# B&R Automation Studio project RTFProj (part 3)

#### Bar_light.c
```c
#include <bur/plctypes.h>
#include <MTBasics.h>
#include <brsystem.h>
#include <math.h>

#ifdef _DEFAULT_INCLUDES
#include <AsDefault.h>
#endif

void resetFB(struct Light *inst);												//Reset basic variables
void PWMControl(struct Light *inst);											//Controls Light in PWM Mode
void BlinkControl(struct Light *inst);											//Allows Blinking of Light

void Light(struct Light *inst)
{
	if ((!inst->Enable) && (inst->internal.MainControlBarLight != INIT_BARLIGHT))//If FB not allowed and switch is not in init state
		inst->internal.MainControlBarLight = DISABLED_BARLIGHT;					//Change state to DISABLED

	switch (inst->internal.MainControlBarLight)									//Main switch controls whole FB
	{
		case INIT_BARLIGHT:														//Check parameter for PWM
			inst->internal.TaskClass.RTInfo_0.enable = 1;
			RTInfo(&inst->internal.TaskClass.RTInfo_0);
			if (!(inst->internal.TaskClass.RTInfo_0.status) && (inst->internal.TaskClass.RTInfo_0.cycle_time > 0))
			{
				if (inst->internal.TaskClass.RTInfo_0.cycle_time <= 1000)
				{
					inst->isPWMEnabled = inst->internal.PWM.PWMEnabled = 1;
					inst->isPWMEnabled = inst->internal.PWM.PWM.Enable = 1;
					inst->internal.PWM.PWM.MinPulseWidth = 0.0008;
					inst->internal.PWM.PWM.Period = 0.008;
					inst->internal.PWM.PWM.Mode = mtBASICS_PULSE_BEGINNING;
				}
				else
					inst->isPWMEnabled = inst->internal.PWM.PWMEnabled = 0;

				inst->internal.PWM.PWM.DutyCycle = 100;
				inst->internal.TaskClass.RTInfo_0.enable = 0;
				inst->internal.TaskClass.CyclicTime = ((inst->internal.TaskClass.RTInfo_0.cycle_time)/800);
				inst->internal.MainControlBarLight = DISABLED_BARLIGHT;
			}
			break;

		case DISABLED_BARLIGHT:
			if (inst->Enable)
			{
				if (inst->DO9322.ModuleOK)
				{
					inst->internal.MainControlBarLight = ENABLED_BARLIGHT;
					resetFB(inst);
				}
				else
				{
					inst->Status = DO9322_NOT_CONNECTED;
					inst->internal.MainControlBarLight = ERROR_BARLIGHT;
				}
			}
			inst->isPowerOn = 0;
			break;

		case ENABLED_BARLIGHT:
			inst->Active = 1;
			if (inst->PowerOn)
			{
				if (inst->Blinking.StartBlinking)
				{
					BlinkControl(inst);
				}
				else if (inst->internal.PWM.PWMEnabled)
				{
					PWMControl(inst);
				}
				else inst->DO9322.DigitalOutput = 1;
				inst->isPowerOn = 1;
			}

			else{
				inst->DO9322.DigitalOutput = 0;
				inst->isPowerOn = 0;
			}
			break;

		case ERROR_BARLIGHT:
			inst->Error = 1;
			break;
	}
}

void resetFB(struct Light *inst)
{
	inst->Active = 0;
	inst->Blinking.StartBlinking = 0;
	inst->DO9322.DigitalOutput = 0;
	inst->DutyCycle = 100;
	inst->Error = 0;
	inst->isPowerOn = 0;
	inst->Status = ERR_OK;
}

void PWMControl(struct Light *inst)
{
	inst->internal.PWM.PWM.DutyCycle = inst->DutyCycle;
	MTBasicsPWM(&inst->internal.PWM.PWM);
	inst->DO9322.DigitalOutput = inst->internal.PWM.PWM.Out;
}

void BlinkControl(struct Light *inst)
{
	inst->internal.BlinkingCounter += 1;
	if ((inst->internal.BlinkingCounter*inst->internal.TaskClass.CyclicTime) < inst->Blinking.BlinkingTime_ms)
	{
		if ((inst->internal.BlinkCounter*inst->internal.TaskClass.CyclicTime) >= inst->Blinking.BlinkPeriod_ms)
		{
			inst->DO9322.DigitalOutput = !inst->DO9322.DigitalOutput;
			inst->internal.BlinkCounter = 0;
		}
		else
		{
			inst->internal.BlinkCounter += 1;
		}
	}
	else
	{
		inst->internal.BlinkingCounter = 0;
		inst->internal.BlinkCounter = 0;
		inst->DO9322.DigitalOutput = 0;
		inst->Blinking.StartBlinking = 0;
	}
}
```

#### Types.typ - Exported data types
```iecst
TYPE
	MainControlBarLight_enum :
		(
		INIT_BARLIGHT := 0,
		DISABLED_BARLIGHT := 1,
		ENABLED_BARLIGHT := 2,
		ERROR_BARLIGHT := 100
		);
	DO9322_type : 	STRUCT
		ModuleOK : BOOL;
		DigitalOutput : BOOL;
	END_STRUCT;
	PWM_type : 	STRUCT
		PWMEnabled : BOOL;
		PWM : MTBasicsPWM;
	END_STRUCT;
	internal_type : 	STRUCT
		init : BOOL;
		TaskClass : TaskClass_type;
		PWM : PWM_type;
		BlinkTime : UINT;
		MainControlBarLight : MainControlBarLight_enum;
		BlinkingCounter : UINT;
		BlinkCounter : UINT;
	END_STRUCT;
	Blink_type : 	STRUCT
		StartBlinking : BOOL;
		BlinkPeriod_ms : UINT;
		BlinkingTime_ms : UINT;
	END_STRUCT;
	TaskClass_type : 	STRUCT
		CyclicTime : UINT;
		RTInfo_0 : RTInfo;
	END_STRUCT;
END_TYPE
```

#### Constants.var - Exported constants
```iecst
VAR CONSTANT
	DO9322_NOT_CONNECTED : UINT := 62150; (*DO module in not connected*)
END_VAR
```

#### Bar_Light.fun - Exported functions and function blocks
```iecst
FUNCTION_BLOCK Light
	VAR_INPUT
		Enable : BOOL;
		DO9322 : DO9322_type;
		PowerOn : BOOL;
		DutyCycle : USINT; (*Power of Light in % [0-100]*)
		Blinking : Blink_type;
	END_VAR
	VAR_OUTPUT
		Active : BOOL;
		Error : BOOL;
		Status : UINT;
		isPWMEnabled : BOOL;
		isPowerOn : BOOL;
	END_VAR
	VAR
		internal : internal_type;
	END_VAR
END_FUNCTION_BLOCK
```

### Data object Logical/ACP10_ETXEN/acp10etxen (Ett)

- acp10etxen.ett (not shown)

### Program Logical/Simulation/Technology/simulation (ANSIC) - Roman Parák program for simulation.

#### simulation.c - Init, cyclic, exit code
```c
/*********************************************************************************************
* B&R Automation - Perfection in Automation (https://www.br-automation.com)
    ******************************************************************************************
    * Program 	    : Master's Thesis - Soccer Table (Simulation)
    * Author  	    : Roman Parak
    * Created 	    : date ...
	* University    : Brno University of Technology(BUT)
	* Faculty       : Faculty of Mechanical Engineering(FME)
	* Study Program : Applied Computer Science and Control
	* Institute     : Institute of Automation and Computer Science
**********************************************************************************************
* Implementation OF PROGRAM simulation(Simulation/Technology/simulation/Program/simulation.c)
**********************************************************************************************/

/*************************** LIBRARIES *********************************/
#include <bur/plc.h>
#include <bur/plctypes.h>
#include <astime.h>
#include <math.h>

#include "rp_funcx1.h"
#include "Structures/simulation_str.h"
#include "Functions/sim_mapp.h"

#ifdef _DEFAULT_INCLUDES
	#include <AsDefault.h>
#endif

/*************************** DEFINITIONS *******************************/
#define EACH_FORMATION 1;

/************************ LOCAL VARIABLES ******************************/

// struct - rp_funcx1
_LOCAL struct forecast_direction f_d;
_LOCAL struct calculation_posDummies c_ppd;
_LOCAL struct calculation_crossingBall c_cb[2];
_LOCAL struct calculation_displacementOfAxes c_doa;
_LOCAL struct start_rotaryAxis start_rotaryAxis_0;
_LOCAL struct control_temperature c_temp;
_LOCAL struct axes_control axes_control_0[4];
_LOCAL struct ball_shooting ball_s;
_LOCAL struct check_attack_mode check_attack_mode_0;
_LOCAL struct start_virtualAxis s_virtualA;
// struct - MpAlarmX
_LOCAL MpAlarmXListUIConnectType AlarmListUI_ConnectType;
_LOCAL MpAlarmXHistoryUIConnectType AlarmHistoryUI_ConnectType;
// udint
_LOCAL UDINT alarm_device_address, specific_directionOfBall;
// usint
_LOCAL USINT max_numberOfFormation;
_LOCAL USINT i_axisNum;
_LOCAL USINT i_bs;
_LOCAL USINT i_ppd, i_ccd, i_ccdCPU, i_ccdHUM, i_cdoa1, i_cdoa2, i_cdoa3;
_LOCAL USINT c_dp;
_LOCAL USINT i_def, i_dp1, i_dp2;
_LOCAL USINT c_bState;
// bool
_LOCAL BOOL ESTOP,error_s,reset_safetyESTOP;
_LOCAL BOOL start_game;
// real
_LOCAL REAL x_posOfCPU[4];
_LOCAL REAL x_posOfHUM[4];
// OUPTUT from the SENSOR & CAMERA
_LOCAL REAL ball1[2], ball2[2], time_B2B;
_LOCAL REAL optical_sensor[4];
_LOCAL REAL reflex_sensor[4];
// state machine
_LOCAL soccer_table_ENUM SOCCER_TABLE_STEP;
_LOCAL soccer_table_ENUM BEFORE_STATE;

/**********************************************************************************************************/
/********************************************** INIT PROGRAM **********************************************/
/**********************************************************************************************************/
void _INIT ProgramInit(void)
{
    /*********************************** declaration variables **********************************/
    // generally
    max_numberOfFormation = 4;
    // axis type -> MAPP
    // linear
	gLinkAxes_linear[0] = gk_mappAxisLS;
    gLinkAxes_linear[1] = df_mappAxisLS;
    gLinkAxes_linear[2] = md_mappAxisLS;
    gLinkAxes_linear[3] = fw_mappAxisLS;
    // rotary
    gLinkAxes_rotary[0] = gk_mappAxisRS;
    gLinkAxes_rotary[1] = df_mappAxisRS;
    gLinkAxes_rotary[2] = md_mappAxisRS;
    gLinkAxes_rotary[3] = fw_mappAxisRS;

    /************************************ control of AlarmX ************************************/
    // adjustment device name
    alarm_device_address = (UDINT) strcpy(mp_alarmX.deviceName_no1_exp,"EXPORT_HISTORY");
    // MpAlarmX Core
    mp_alarmX.mp_core.MpLink         = &gAlarmXCoreS;
    mp_alarmX.mp_core.Enable         = 1;
    // MpAlarmX ListUI
    mp_alarmX.mp_listUI.MpLink       = &gAlarmXCoreS;
    mp_alarmX.mp_listUI.Enable       = 1;
    mp_alarmX.mp_listUI.UIConnect    = &AlarmListUI_ConnectType;
    // MpAlarmX History
    mp_alarmX.mp_history.MpLink      = &gAlarmXHistoryS;
    mp_alarmX.mp_history.Enable      = 1;
    mp_alarmX.mp_history.DeviceName  = &mp_alarmX.deviceName_no1_exp;
    // MpAlarmX HistoryUI
    mp_alarmX.mp_historyUI.MpLink    = &gAlarmXHistoryS;
    mp_alarmX.mp_historyUI.Enable    = 1;
    mp_alarmX.mp_historyUI.UIConnect = &AlarmHistoryUI_ConnectType;

    /************************************* control of axes **************************************/
    for(i_axisNum = 0; i_axisNum <= max_numberOfFormation - 1; i_axisNum++){
        // initialization ACOPOS variables through function(get_axisParam), that returns two variables type of UDINT
        // into the structure -> axesAcopos(have two parameters : linear, rotary)
        axis_acopos = get_axisParam(i_axisNum);
        // linear -> LinMot
        // linear axis basic
        mp_Axis.mp_axisLinear[i_axisNum].Enable     = 1;
        mp_Axis.mp_axisLinear[i_axisNum].MpLink     = &gLinkAxes_linear[i_axisNum];
        mp_Axis.mp_axisLinear[i_axisNum].Parameters = &mp_Axis.param_axisLinear[i_axisNum];
        mp_Axis.mp_axisLinear[i_axisNum].Axis       = axis_acopos.linear;
        // linear cyclic set
        mp_Axis.mp_cyclicSetLinear[i_axisNum].Enable     = 1;
        mp_Axis.mp_cyclicSetLinear[i_axisNum].MpLink     = &gLinkAxes_linear[i_axisNum];
        mp_Axis.mp_cyclicSetLinear[i_axisNum].Parameters = &mp_Axis.param_cyclicSetLinear[i_axisNum];
		// adjustment max velocity
		mp_Axis.param_cyclicSetLinear[i_axisNum].PositionModeMaxVelocity = 30000;
		// config
		mp_Axis.mp_configAxisLinear[i_axisNum].Enable 		 = 1;
		mp_Axis.mp_configAxisLinear[i_axisNum].MpLink 		 = &gLinkAxes_linear[i_axisNum];
		mp_Axis.mp_configAxisLinear[i_axisNum].Configuration = &mp_Axis.param_configAxisLinear[i_axisNum];
        // rotary -> EnDat
        // rotary axis basic
        mp_Axis.mp_axisRotary[i_axisNum].Enable     = 1;
        mp_Axis.mp_axisRotary[i_axisNum].MpLink     = &gLinkAxes_rotary[i_axisNum];
        mp_Axis.mp_axisRotary[i_axisNum].Parameters = &mp_Axis.param_axisRotary[i_axisNum];
        mp_Axis.mp_axisRotary[i_axisNum].Axis       = axis_acopos.rotary;
        // rotary cyclic set
        mp_Axis.mp_cyclicSetRotary[i_axisNum].Enable     = 1;
        mp_Axis.mp_cyclicSetRotary[i_axisNum].MpLink     = &gLinkAxes_rotary[i_axisNum];
        mp_Axis.mp_cyclicSetRotary[i_axisNum].Parameters = &mp_Axis.param_cyclicSetRotary[i_axisNum];
		// adjustment max velocity
		mp_Axis.param_cyclicSetRotary[i_axisNum].PositionModeMaxVelocity = 85000;
		// config
		mp_Axis.mp_configAxisRotary[i_axisNum].Enable 		 = 1;
		mp_Axis.mp_configAxisRotary[i_axisNum].MpLink 		 = &gLinkAxes_rotary[i_axisNum];
		mp_Axis.mp_configAxisRotary[i_axisNum].Configuration = &mp_Axis.param_configAxisRotary[i_axisNum];
		// temperature - linear
		mp_Axis.param_axisLinear[i_axisNum].CyclicRead.MotorTempMode = mpAXIS_READ_POLLING_5s;
		// temperature - rotary
		mp_Axis.param_axisRotary[i_axisNum].CyclicRead.MotorTempMode = mpAXIS_READ_POLLING_5s;
    }
    // initialization switch
    SOCCER_TABLE_STEP = RST_EMPTY;
    // initialization x axes for CPU
    x_posOfCPU[0] = 800;
    x_posOfCPU[1] = 2300;
    x_posOfCPU[2] = 5300;
    x_posOfCPU[3] = 8300;
    // initialization x axes for HUMAN
    x_posOfHUM[0] = 3800;
    x_posOfHUM[1] = 6800;
    x_posOfHUM[2] = 9800;
    x_posOfHUM[3] = 11300;
    // OUPTUT from the SENSOR & CAMERA
    // CAMERA
    ball1[0] = 0;
    ball1[1] = 0;
    ball2[0] = 0;
    ball2[1] = 0;
    time_B2B = 0;
    // SENSOR
    optical_sensor[0] = 0;
    optical_sensor[1] = 0;
    optical_sensor[2] = 0;
    optical_sensor[3] = 0;

    reflex_sensor[0] = 1;
    reflex_sensor[1] = 1;
    reflex_sensor[2] = 1;
    reflex_sensor[3] = 1;
	// init safety
	ESTOP = 1;
	// axes control
	// FB for linear and fotary axes -> Control
	axes_control_0[0].Enable			 = 1;
	axes_control_0[0].linear_axis_cyclic = &mp_Axis.mp_cyclicSetLinear[0];
	axes_control_0[0].linear_axis_param  = &mp_Axis.param_cyclicSetLinear[0];
	axes_control_0[0].rotary_axis_cyclic = &mp_Axis.mp_cyclicSetRotary[0];
	axes_control_0[0].rotary_axis_param  = &mp_Axis.param_cyclicSetRotary[0];

	s_virtualA.Enable 	  = 1;
	s_virtualA.axis_name  = &mp_Axis.mp_axisLinear[0];
	s_virtualA.axis_param = &mp_Axis.param_axisLinear[0];
}// end _INIT

/**********************************************************************************************************/
/********************************************** MAIN PROGRAM **********************************************/
/**********************************************************************************************************/
void _CYCLIC ProgramCyclic(void)
{
    switch(SOCCER_TABLE_STEP){
		case RST_EMPTY:
			{

			}
			break;
		case RST_INITIALIZATION_1:
			{
				// home virtual linear axis
				s_virtualA.start_btn = 1;
				start_virtualAxis(&s_virtualA);

				if(s_virtualA.succesfully == 1 && (mp_Axis.mp_axisLinear[0].PowerOn == 1 && mp_Axis.mp_axisLinear[0].IsHomed == 1)){
					SOCCER_TABLE_STEP = RST_INITIALIZATION_2;
				}
			}
			break;
		case RST_INITIALIZATION_2:
			{

			}
			break;
		case RST_INITIALIZATION_3:
			{

			}
			break;
		case RST_INITIALIZATION_4:
			{
				check_attack_mode_0.ball1_x = ball1[0];
				check_attack_mode_0.ball1_y = ball1[1];
				check_attack_mode_0.ball2_x = ball2[0];
				check_attack_mode_0.ball2_y = ball2[1];

				check_attack_mode_0.act_displacement_cpu[2] = 112;
				check_attack_mode_0.angle_ofRotation[2]     = -250;
				// call function
				check_attack_mode(&check_attack_mode_0);
			}
			break;
        case RST_CALCULATION_DEFENSE:
            {
                // calculation forecast direction
                f_d.ball1_x = ball1[0];
                f_d.ball1_y = ball1[1];
                f_d.ball2_x = ball2[0];
                f_d.ball2_y = ball2[1];
                forecast_direction(&f_d);
                // calculation pos dummies opponent
				// maximum displacement of individual axes
				c_ppd.max_disp[0] = 1000;
				c_ppd.max_disp[0] = 1850;
				c_ppd.max_disp[0] = 650;
				c_ppd.max_disp[0] = 955;
				// minimum displacement of individual axes
				c_ppd.min_disp[0] = -1000;
				c_ppd.min_disp[0] = -1850;
				c_ppd.min_disp[0] = -650;
				c_ppd.min_disp[0] = -955;
                for(i_ppd = 0; i_ppd < (int)(sizeof(optical_sensor)/sizeof(optical_sensor[0])); i_ppd++){
                    c_ppd.displacement[i_ppd] = optical_sensor[i_ppd];
                }

                calculation_posDummies(&c_ppd);
                // calculation crossing ball
                for(i_ccd = 0; i_ccd < (int)(sizeof(ball1)/sizeof(ball1[0])); i_ccd++){
                    c_cb[i_ccd].ball1_x = ball1[0];
                    c_cb[i_ccd].ball1_y = ball1[1];
                    c_cb[i_ccd].ball2_x = ball2[0];
                    c_cb[i_ccd].ball2_y = ball2[1];
                    c_cb[i_ccd].first_reflection_x  = f_d.first_reflectionX;
                    c_cb[i_ccd].first_reflection_y  = f_d.first_reflectionY;
                    c_cb[i_ccd].second_reflection_x = f_d.second_reflectionX;
                    c_cb[i_ccd].second_reflection_y = f_d.second_reflectionY;
                    c_cb[i_ccd].tilted   = f_d.tilted;
                    c_cb[i_ccd].time_B2B = time_B2B;

                    if(i_ccd == 0){
                        for(i_ccdCPU = 0; i_ccdCPU < (int)(sizeof(x_posOfCPU)/sizeof(x_posOfCPU[0])); i_ccdCPU++){
                            c_cb[i_ccd].x_positions[i_ccdCPU] = x_posOfCPU[i_ccdCPU];
                        }
                    }else if(i_ccd == 1){
                        for(i_ccdHUM = 0; i_ccdHUM < (int)(sizeof(x_posOfHUM)/sizeof(x_posOfHUM[0])); i_ccdHUM++){
                            c_cb[i_ccd].x_positions[i_ccdHUM] = x_posOfHUM[i_ccdHUM];
                        }
                    }
                    calculation_crossingBall(&c_cb[i_ccd]);
                }
                // calculation displacement
                c_doa.tilted             = f_d.tilted;
                specific_directionOfBall = (UDINT) strcpy(c_doa.specific_direction,f_d.specific_direction);
                for(i_cdoa1 = 0; i_cdoa1 < (int)(sizeof(c_cb[1].count_axesIntersection)/sizeof(c_cb[1].count_axesIntersection[0])); i_cdoa1++){
                    c_doa.count_axesIntersectionHUM[i_cdoa1] = c_cb[1].count_axesIntersection[i_cdoa1];
                }
                for(i_cdoa2 = 0; i_cdoa2 < (int)(sizeof(c_cb[0].act_posOfAxesY)/sizeof(c_cb[0].act_posOfAxesY[0])); i_cdoa2++){
                    c_doa.act_posOfAxesCPU_Y[i_cdoa2]    = c_cb[0].act_posOfAxesY[i_cdoa2];
                    c_doa.time_axisIntersection[i_cdoa2] = c_cb[0].time_axisIntersection[i_cdoa2];
                    c_doa.act_displacementCPU[i_cdoa2]   = 0; // actual displacement
                    c_doa.reversed_HUM[i_cdoa2]          = reflex_sensor[i_cdoa2];
                }
                c_doa.act_posOfAxesHUM_Y[0] = c_cb[1].act_posOfAxesY[3];
                c_doa.act_posOfAxesHUM_Y[1] = c_cb[1].act_posOfAxesY[2];
                c_doa.act_posOfAxesHUM_Y[2] = c_cb[1].act_posOfAxesY[1];
                c_doa.act_posOfAxesHUM_Y[3] = c_cb[1].act_posOfAxesY[0];
                for(i_cdoa3 = 0; i_cdoa3 < (int)(sizeof(c_ppd.actual_positionsOfDummies)/sizeof(c_ppd.actual_positionsOfDummies[0])); i_cdoa3++){
                    c_doa.act_posOfDummiesH[i_cdoa3] = c_ppd.actual_positionsOfDummies[i_cdoa3];
                }
                c_doa.x_posOfBall[0] = ball1[0];
                c_doa.x_posOfBall[1] = ball2[0];
                calculation_displacementOfAxes(&c_doa);

				for(i_def = 0; i_def <= max_numberOfFormation - 1; i_def++){
					if(!isnan(c_doa.velocity[i_def])){
						axes_control_0[i_def].linear_param.acceleration = c_doa.acceleration[i_def];
						axes_control_0[i_def].linear_param.deceleration = c_doa.deceleration[i_def];
						axes_control_0[i_def].linear_param.velocity     = c_doa.velocity[i_def];
						axes_control_0[i_def].linear_param.displacement = c_doa.displacement[i_def];
					}
				}

				/*
				if(ESTOP == 0){
					SOCCER_TABLE_STEP = RST_SAFETY;
				}else{
					c_dp = 0;

					if(c_dp == 0){
						SOCCER_TABLE_STEP = RST_MOVE_INTO_DEFENSE_POS1;
					}
				}
				*/
            }
            break;
		case RST_MOVE_INTO_DEFENSE_POS1:
			{
				for(i_dp1 = 0; i_dp1 <= max_numberOfFormation - 1; i_dp1++){
					axes_control_0[i_dp1].start_move = 1;
				}

				if(ESTOP == 0){
					SOCCER_TABLE_STEP = RST_SAFETY;
				}else{
					SOCCER_TABLE_STEP = RST_MOVE_INTO_DEFENSE_POS2;
				}
			}
			break;
		case RST_MOVE_INTO_DEFENSE_POS2:
			{
				for(i_dp2 = 0; i_dp2 <= max_numberOfFormation - 1; i_dp2++){
					if(axes_control_0[i_dp2].successfully == 1){
						axes_control_0[i_dp2].start_move = 0;
						c_dp++;
					}
				}

				if(ESTOP == 0){
					SOCCER_TABLE_STEP = RST_SAFETY;
				}else{
					if(c_dp == max_numberOfFormation){
						SOCCER_TABLE_STEP = RST_INITIALIZATION_4;
					}
				}
			}
		case RST_SAFETY:
			{
			}
			break;
		case RST_AFTER_SAFETY:
			{

			}
			break;
    }// end switch

    /************************** call function & function blocks **************************/
    // AlarmX
    MpAlarmXCore(&mp_alarmX.mp_core);
    MpAlarmXListUI(&mp_alarmX.mp_listUI);
    MpAlarmXHistory(&mp_alarmX.mp_history);
    MpAlarmXHistoryUI(&mp_alarmX.mp_historyUI);
    // Active AxisBasic & AxisCyclicSet -> through the individual functions
    start_axesBasic(max_numberOfFormation,&mp_Axis.mp_axisLinear,&mp_Axis.mp_axisRotary);
    start_axesCyclic(max_numberOfFormation,&mp_Axis.mp_cyclicSetLinear,&mp_Axis.mp_cyclicSetRotary);

	// control temperature
	//control_temperature(&c_temp);
	if(SOCCER_TABLE_STEP >= 3){
		axes_control(&axes_control_0[0]);
	}

}// end _CYCLIC
```

#### simulation_str.h
```c
/*********************************************************************************************
* B&R Automation - Perfection in Automation (https://www.br-automation.com)
    ******************************************************************************************
    * Program 	    : Master's Thesis - Soccer Table (Simulation)
    * Author  	    : Roman Parak
    * Created 	    : date ...
	* University    : Brno University of Technology(BUT)
	* Faculty       : Faculty of Mechanical Engineering(FME)
	* Study Program : Applied Computer Science and Control
	* Institute     : Institute of Automation and Computer Science
**********************************************************************************************
* Implementation OF PROGRAM simulation(Simulation/Technology/simulation/Structures/simulation_str.h)
**********************************************************************************************/

/*************************** LIBRARIES *********************************/
#include <bur/plc.h>
#include <bur/plctypes.h>
#include <AsString.h>
#include <AsWStr.h>

#ifdef _DEFAULT_INCLUDES
    #include <AsDefault.h>
#endif

/**********************************************************************************************************/
/************************************** STRUCTURE TYPE ****************************************************/
/**********************************************************************************************************/

/***************************************** sim_mapp.h *****************************************************/
/***************************** ALARM ***********************************/
typedef struct mappAlarmX_STR{
    // list
    struct MpAlarmXCore   mp_core;
    struct MpAlarmXListUI mp_listUI;
    // history
    struct    MpAlarmXHistory mp_history;
    struct    MpAlarmXHistoryUI mp_historyUI;
    plcstring deviceName_no1_exp[21];
} mappAlarmX_STR;

/***************************** AXIS ************************************/
typedef struct mappAxisBasic_STR{
	// === Linear Axes === //
	// axis basic
	struct MpAxisBasic        mp_axisLinear[4];
	struct MpAxisBasicParType param_axisLinear[4];
	// cyclic set
	struct MpAxisCyclicSet        mp_cyclicSetLinear[4];
	struct MpAxisCyclicSetParType param_cyclicSetLinear[4];
	// config
	struct MpAxisBasicConfig mp_configAxisLinear[4];
	struct MpAxisBasicConfigType param_configAxisLinear[4];
	// === Rotary Axes === //
	// axis basic
	struct MpAxisBasic        mp_axisRotary[4];
	struct MpAxisBasicParType param_axisRotary[4];
	// cyclic set
	struct MpAxisCyclicSet        mp_cyclicSetRotary[4];
	struct MpAxisCyclicSetParType param_cyclicSetRotary[4];
	// config
	struct MpAxisBasicConfig mp_configAxisRotary[4];
	struct MpAxisBasicConfigType param_configAxisRotary[4];
} mappAxisBasic_STR;

/***************************** GET AXIS PARAM. ************************************/
typedef struct axesAcopos{
    UDINT linear;
    UDINT rotary;
}axesAcopos;

/*********************************** sim_forecast_direction.h *********************************************/
/***************************** FORECAST DIR.. ************************************/
typedef struct forecastDirection{
	BOOL direction;
	INT first_reflectX;
	INT first_reflectY;
	INT second_reflectX;
	INT second_reflectY;
	plcstring specific_direction[30];
}forecastDirection;
/***************************** CALC. DIR. OF TILT **********************************/
typedef struct tiltDirection{
	INT first_reflectX;
	INT first_reflectY;
	INT state_ofDirection;
    plcstring specific_direction[10];
}tiltDirection;
/***************************** CALC. NEXT DIR. *************************************/
typedef struct nextDirection{
	INT second_reflectX;
	INT second_reflectY;
}nextDirection;

/**********************************************************************************************************/
/**************************************** GLOBAL VARIABLES ************************************************/
/**********************************************************************************************************/

/***************************************** sim_mapp.h *****************************************************/
// my structures
_GLOBAL mappAlarmX_STR mp_alarmX;
_GLOBAL mappAxisBasic_STR mp_Axis;
_GLOBAL axesAcopos axis_acopos;

// axis type -> ACOPOS
// goalkeeper
_GLOBAL ACP10AXIS_typ gkLinS;
_GLOBAL ACP10AXIS_typ gkRotS;
// defender
_GLOBAL ACP10AXIS_typ dfLinS;
_GLOBAL ACP10AXIS_typ dfRotS;
// midfielder
_GLOBAL ACP10AXIS_typ mdLinS;
_GLOBAL ACP10AXIS_typ mdRotS;
// forward
_GLOBAL ACP10AXIS_typ fwLinS;
_GLOBAL ACP10AXIS_typ fwRotS;
// axis type -> MAPP
_GLOBAL struct MpComIdentType gLinkAxes_rotary[4];
_GLOBAL struct MpComIdentType gLinkAxes_linear[4];

/**********************************************************************************************************/
/************************************** FUNCTIONS & FUNCTIONS BLOCKS **************************************/
/**********************************************************************************************************/
void start_axesBasic(USINT num_ofAxes,struct MpAxisBasic* axis_linear,struct MpAxisBasic* axis_rotary);
void start_axesCyclic(USINT num_ofAxes,struct MpAxisCyclicSet* cyclic_linear,struct MpAxisCyclicSet* cyclic_rotary);
struct axesAcopos get_axisParam(int idx_ofIteration);
```

#### sim_mapp.h
```c
/*********************************************************************************************
* B&R Automation - Perfection in Automation (https://www.br-automation.com)
    ******************************************************************************************
    * Program 	    : Master's Thesis - Soccer Table (Simulation)
    * Author  	    : Roman Parak
    * Created 	    : date ...
	* University    : Brno University of Technology(BUT)
	* Faculty       : Faculty of Mechanical Engineering(FME)
	* Study Program : Applied Computer Science and Control
	* Institute     : Institute of Automation and Computer Science
**********************************************************************************************
* Implementation OF PROGRAM simulation(Simulation/Technology/simulation/Functions/sim_mapp.h)
**********************************************************************************************/

/*************************** LIBRARIES *********************************/
#include <bur/plc.h>
#include <bur/plctypes.h>
#include <AsString.h>
#include <AsWStr.h>

#ifdef _DEFAULT_INCLUDES
    #include <AsDefault.h>
#endif

/**********************************************************************************************************/
/************************************** FUNCTIONS & FUNCTIONS BLOCKS **************************************/
/**********************************************************************************************************/
void start_axesBasic(USINT num_ofAxes,struct MpAxisBasic* axis_linear,struct MpAxisBasic* axis_rotary){
    int i;
    // Axis Basic
    // function to start the individual axes
    // the cycle is carried out through number of axes
    for(i = 0; i <= num_ofAxes - 1; i++){
        // mapp axis basic
        MpAxisBasic(&axis_linear[i]);
        MpAxisBasic(&axis_rotary[i]);
    }
}

void start_axesCyclic(USINT num_ofAxes,struct MpAxisCyclicSet* cyclic_linear,struct MpAxisCyclicSet* cyclic_rotary){
    int i;
    // Axis Cyclic Set
    // function to start the individual axes
    // the cycle is carried out through number of axes
    for(i = 0; i <= num_ofAxes - 1; i++){
        // mapp axis cyclic set
        MpAxisCyclicSet(&cyclic_linear[i]);
        MpAxisCyclicSet(&cyclic_rotary[i]);
    }
}

struct axesAcopos get_axisParam(int idx_ofIteration){
    // input into the function is number of iteration(in the init part)
    // create auxiliary structures and enumeration type(for state machine)
    struct axesAcopos a;
    typedef enum {aNUM1 = 0, aNUM2, aNUM3, aNUM4}wState_ofAxes;
    wState_ofAxes new_idx; // initialize state machine
    new_idx = idx_ofIteration;
    // gradually into the state machine loading indexes from initialization part
    // each state of machine has initialization both engines linear and rotary, on its own axis
    // output of this function is structure, that has two parameters(linear,rotary axis)
    switch(new_idx){
        case aNUM1:
            // goalkeeper
            a.linear = &gkLinS;
            a.rotary = &gkRotS;
            return a;
            break;
        case aNUM2:
            // defender
            a.linear = &dfLinS;
            a.rotary = &dfRotS;
            return a;
            break;
        case aNUM3:
            // midfielder
            a.linear = &mdLinS;
            a.rotary = &mdRotS;
            return a;
            break;
        case aNUM4:
            // forward
            a.linear = &fwLinS;
            a.rotary = &fwRotS;
            break;
    }
}
```

### Program Logical/Simulation/Technology/sim_cam_sens_sd_s (ANSIC) - Lubo,Radek program for simulation.

#### main_sim.c - Init, cyclic, exit code
```c
/*********************************************************************************************
* B&R Automation - Perfection in Automation (https://www.br-automation.com)
    ******************************************************************************************
    * Program 	    : Bachelor's Thesis
    * Author  	    : Lubo Bubco, Radek Otradovský
    * Created 	    : date ...
	* University    : Brno University of Technology(BUT)
	* Faculty       : Faculty of Mechanical Engineering(FME), Faculty of Electrical Engineering and Communication(FEEC)
**********************************************************************************************
* Implementation OF PROGRAM sim_cam_sens_sd_s(Simulation/Technology/sim_cam_sens_sd_s/main_sim.c)
**********************************************************************************************/

#include <bur/plctypes.h>
#include <string.h>
#include <math.h>
#include "rp_funcx1.h"

#ifdef _DEFAULT_INCLUDES
	#include <AsDefault.h>
#endif

_LOCAL struct measurement_ofScore measurement_ofScore_1;

void _INIT ProgramInit(void)
{

}

void _CYCLIC ProgramCyclic(void)
{
    measurement_ofScore(&measurement_ofScore_1);
}
```


- Data object Logical/Simulation/Motion/dfRotSobj/dfRotSa (Apt) (no source held here)

- Data object Logical/Simulation/Motion/dfRotSobj/dfRotSi (Ax) (no source held here)

- Data object Logical/Simulation/Motion/gkRotSobj/gkRotSa (Apt) (no source held here)

- Data object Logical/Simulation/Motion/gkRotSobj/gkRotSi (Ax) (no source held here)

- Data object Logical/Simulation/Motion/dfLinSobj/dfLinSa (Apt) (no source held here)

- Data object Logical/Simulation/Motion/dfLinSobj/dfLinSi (Ax) (no source held here)

- Data object Logical/Simulation/Motion/gkLinSobj/gkLinSa (Apt) (no source held here)

- Data object Logical/Simulation/Motion/gkLinSobj/gkLinSi (Ax) (no source held here)

### Package Logical/Simulation/Motion/fwRotSobj - fwRotSobj

### Data object Logical/Simulation/Motion/fwRotSobj/fwRotSa (Apt)

#### fwRotSa.apt
```
AcoposParameterTable:
  Root Parameters
```

- Data object Logical/Simulation/Motion/fwRotSobj/fwRotSi (Ax) (no source held here)

- Data object Logical/Simulation/Motion/mdRotSobj/mdRotSa (Apt) (no source held here)

- Data object Logical/Simulation/Motion/mdRotSobj/mdRotSi (Ax) (no source held here)

### Package Logical/Simulation/Motion/fwLinSobj - fwLinSobj

- Data object Logical/Simulation/Motion/fwLinSobj/fwLinSa (Apt) (no source held here)

### Data object Logical/Simulation/Motion/fwLinSobj/fwLinSi (Ax)

#### fwLinSi.ax
```
InitParameter (Version=3.16.2, NcSwId=Acp10)
  ACP10AXIS_typ:
    dig_in:
      level:
        reference = ncACTIV_HI
        pos_hw_end = ncACTIV_HI
        neg_hw_end = ncACTIV_HI
        trigger1 = ncACTIV_HI
        trigger2 = ncACTIV_HI
    encoder_if:
      parameter:
        count_dir = ncSTANDARD
        scaling:
          load:
            units = 1000
            rev_motor = 1
    limit:
      parameter:
        v_pos = 10000
        v_neg = 10000
        a1_pos = 50000
        a2_pos = 50000
        a1_neg = 50000
        a2_neg = 50000
        t_jolt = 0
        t_in_pos = 0
        pos_sw_end = 2000000000
        neg_sw_end = -2000000000
        ds_warning = 500
        ds_stop = 1000
        a_stop = 1.0e30
        dv_stop = 0
        dv_stop_mode = ncOFF
    controller:
      mode = ncPOSITION
      position:
        kv = 50
        tn = 0
        t_predict = 0.0004
        t_total = 0.0004
        p_max = 1.0e30
        i_max = 0
      speed:
        kv = 2.0
        tn = 0
        t_filter = 0.0
        isq_filter1:
          type = ncOFF
          a0 = 0.0
          a1 = 0.0
          b0 = 0.0
          b1 = 0.0
          b2 = 0.0
          c0_par_id = 0
          c1_par_id = 0
        isq_filter2:
          type = ncOFF
          a0 = 0.0
          a1 = 0.0
          b0 = 0.0
          b1 = 0.0
          b2 = 0.0
          c0_par_id = 0
          c1_par_id = 0
        isq_filter3:
          type = ncOFF
          a0 = 0.0
          a1 = 0.0
          b0 = 0.0
          b1 = 0.0
          b2 = 0.0
          c0_par_id = 0
          c1_par_id = 0
      uf:
        type = ncLINEAR
        auto_config = ncMOTOR_PAR
        u0 = 0
        un = 0
        fn = 50.0
        k_f_slip = 0
      ff:
        torque_load = 0.0
        torque_pos = 0.0
        torque_neg = 0.0
        kv_torque = 0.0
        inertia = 0.0
        t_filter_a = 0.0
    move:
      stop:
        parameter[0]:
          decel_ramp = ncA_LIMIT
          controller = ncON
        parameter[1]:
          decel_ramp = ncA_LIMIT
          controller = ncON
        parameter[2]:
          decel_ramp = ncA_LIMIT
          controller = ncON
        parameter[3]:
          decel_ramp = ncA_LIMIT
          controller = ncON
        quickstop:
          decel_ramp = ncA_LIMIT
        drive_error:
          decel_ramp = ncA_LIMIT
      homing:
        parameter:
          s = 0
          v_switch = 5000
          v_trigger = 500
          a = 50000
          mode = ncDIRECT
          edge_sw = ncPOSITIVE
          start_dir = ncPOSITIVE
          trigg_dir = ncPOSITIVE
          ref_pulse = ncOFF
          fix_dir = ncOFF
          tr_s_block = 0
          torque_lim = 0
          ds_block = 0
          ds_stop = 0
      basis:
        parameter:
          v_pos = 5000
          v_neg = 5000
          a1_pos = 50000
          a2_pos = 50000
          a1_neg = 50000
          a2_neg = 50000
    message:
      text:
        parameter:
          format = ncBREAK
          columns = 80
          data_modul = acp10etxen
```


- Data object Logical/Simulation/Motion/mdLinSobj/mdLinSa (Apt) (no source held here)

- Data object Logical/Simulation/Motion/mdLinSobj/mdLinSi (Ax) (no source held here)

### Package Logical/Real_Game/Motion/rotaryFWobj - rotaryFWobj

- Data object Logical/Real_Game/Motion/rotaryFWobj/rotaryFWa (Apt) (no source held here)

### Data object Logical/Real_Game/Motion/rotaryFWobj/rotaryFWi (Ax)

#### rotaryFWi.ax
```
InitParameter (Version=3.16.2, NcSwId=ACP10)
  ACP10AXIS_typ:
    dig_in:
      level:
        reference = ncACTIV_HI
        pos_hw_end = ncACTIV_HI
        neg_hw_end = ncACTIV_HI
        trigger1 = ncACTIV_HI
        trigger2 = ncACTIV_HI
    encoder_if:
      parameter:
        count_dir = ncSTANDARD
        scaling:
          load:
            units = 3600
            rev_motor = 1
    limit:
      parameter:
        v_pos = 100000.0
        v_neg = 100000.0
        a1_pos = 4000000.0
        a2_pos = 4000000.0
        a1_neg = 4000000.0
        a2_neg = 4000000.0
        t_jolt = 0.04
        t_in_pos = 0.0
        pos_sw_end = 3601
        neg_sw_end = -3601
        ds_warning = 30.0
        ds_stop = 170.0
        a_stop = 1.0E+30
        dv_stop = 0.0
        dv_stop_mode = ncOFF
    controller:
      mode = ncPOSITION + ncFF
      position:
        kv = 320.0
        tn = 0.0
        t_predict = 0.0004
        t_total = 0.0004
        p_max = 1.0E+30
        i_max = 0.0
      speed:
        kv = 1.1
        tn = 0.0
        t_filter = 0.0
        isq_filter1:
          type = ncNOTCH
          a0 = 2338.55
          a1 = 400.0
          b0 = 0.0
          b1 = 0.0
          b2 = 0.0
          c0_par_id = 0
          c1_par_id = 0
        isq_filter2:
          type = ncOFF
          a0 = 0.0
          a1 = 0.0
          b0 = 0.0
          b1 = 0.0
          b2 = 0.0
          c0_par_id = 0
          c1_par_id = 0
        isq_filter3:
          type = ncOFF
          a0 = 0.0
          a1 = 0.0
          b0 = 0.0
          b1 = 0.0
          b2 = 0.0
          c0_par_id = 0
          c1_par_id = 0
      uf:
        type = ncLINEAR
        auto_config = ncMOTOR_PAR
        u0 = 0.0
        un = 0.0
        fn = 50.0
        k_f_slip = 0.0
      ff:
        torque_load = 0.0
        torque_pos = 0.043882
        torque_neg = 0.037949
        kv_torque = 0.00362983
        inertia = 0.000102625
        t_filter_a = 0.0
    move:
      stop:
        parameter[0]:
          decel_ramp = ncA_LIMIT
          controller = ncON
        parameter[1]:
          decel_ramp = ncA_LIMIT
          controller = ncON
        parameter[2]:
          decel_ramp = ncA_LIMIT
          controller = ncON
        parameter[3]:
          decel_ramp = ncA_LIMIT
          controller = ncON
        quickstop:
          decel_ramp = ncA_LIMIT
        drive_error:
          decel_ramp = ncA_LIMIT
      homing:
        parameter:
          s = 0
          v_switch = 50.0
          v_trigger = 5.0
          a = 500.0
          mode = ncDIRECT
          edge_sw = ncPOSITIVE
          start_dir = ncPOSITIVE
          trigg_dir = ncPOSITIVE
          ref_pulse = ncOFF
          fix_dir = ncOFF
          tr_s_block = 0.0
          torque_lim = 0.0
          ds_block = 0.0
          ds_stop = 0.0
      basis:
        parameter:
          v_pos = 84000.0
          v_neg = 84000.0
          a1_pos = 3850000.0
          a2_pos = 3850000.0
          a1_neg = 3850000.0
          a2_neg = 3850000.0
    message:
      text:
        parameter:
          format = ncBREAK + ncZERO
          columns = 80
          data_modul = acp10etxen
```

### Package Logical/Real_Game/Motion/rotaryMDobj - rotaryMDobj

### Data object Logical/Real_Game/Motion/rotaryMDobj/rotaryMDa (Apt)

#### rotaryMDa.apt
```
AcoposParameterTable:
  Root Parameters:
    719 = 1 (Name=ENCOD_CMD)  // Encoder1: Encoder command
```

- Data object Logical/Real_Game/Motion/rotaryMDobj/rotaryMDi (Ax) (no source held here)

### Package Logical/Real_Game/Motion/linearFWobj - linearFWobj

### Data object Logical/Real_Game/Motion/linearFWobj/linearFWa (Apt)

#### linearFWa.apt
```
AcoposParameterTable:
  Root Parameters:
    linMot__PS01_23x80.xml:
      LinMot: PS01-23x80/150x210  // Version: 1.1
        Motor (Disabled=FALSE)
          30 = 0x0002 (Name=MOTOR_TYPE, Disabled=FALSE)  // Motor: Type
          31 = 0x0203 (Name=MOTOR_COMPATIBILITY, Disabled=FALSE)  // Motor: Software compatibility
          46 = 1 (Name=MOTOR_WIND_CONNECT, Disabled=FALSE)  // Motor: Winding connection
          47 = 1 (Name=MOTOR_POLEPAIRS, Disabled=FALSE)  // Motor: Number of pole-pairs
          1208 = 2 (Name=MOTOR_NUM_PHASES)  // Motor: Number of motor phases
          48 = 72 (Name=MOTOR_VOLTAGE_RATED, Unit=V, Disabled=FALSE)  // Motor: Rated voltage
          49 = 5.209 (Name=MOTOR_VOLTAGE_CONST, Unit=mV*min, Disabled=FALSE)  // Motor: Voltage constant
          51 = 18000 (Name=MOTOR_SPEED_MAX, Unit=1/min, Disabled=FALSE)  // Motor: Maximum speed
          54 = 0.14 (Name=MOTOR_TORQ_MAX, Unit=Nm, Disabled=FALSE)  // Motor: Peak torque
          55 = 0.035 (Name=MOTOR_TORQ_CONST, Unit=Nm/A, Disabled=FALSE)  // Motor: Torque constant
          58 = 4 (Name=MOTOR_CURR_MAX, Unit=A, Disabled=FALSE)  // Motor: Peak current
          60 = 12.5 (Name=MOTOR_STATOR_RESISTANCE, Unit=Ohm, Disabled=FALSE)  // Motor: Stator resistance
          61 = 0.0014 (Name=MOTOR_STATOR_INDUCTANCE, Unit=Henry, Disabled=FALSE)  // Motor: Stator inductance
          62 = 0.0000027 (Name=MOTOR_INERTIA, Unit=kgmp, Disabled=FALSE)  // Motor: Moment of inertia
          63 = 1.5707963 (Name=MOTOR_COMMUT_OFFSET, Unit=rad, Disabled=FALSE)  // Motor: Commutation offset
          276 = 4 (Name=PHASING_MODE, Disabled=FALSE)  // Motor: Phasing: Mode
        50 = 18000 (Name=MOTOR_SPEED_RATED, Unit=1/min, Disabled=FALSE)  // Motor: Rated speed
        Temperature model (Disabled=FALSE)
          56 = 0.82 (Name=MOTOR_CURR_STALL, Unit=A, Disabled=FALSE)  // Motor: Stall current
          57 = 0.82 (Name=MOTOR_CURR_RATED, Unit=A, Disabled=FALSE)  // Motor: Rated current
          52 = 0.03 (Name=MOTOR_TORQ_STALL, Unit=Nm, Disabled=FALSE)  // Motor: Stall torque
          53 = 0.03 (Name=MOTOR_TORQ_RATED, Unit=Nm, Disabled=FALSE)  // Motor: Rated torque
          59 = 0.11 (Name=MOTOR_WIND_CROSS_SECT, Unit=mmp, Disabled=FALSE)  // Motor: Line cross section
          849 = 135.72 (Name=MOTOR_TAU_THERM, Unit=s, Disabled=FALSE)  // Motor: Thermal time constant
          74 = 110 (Name=MOTOR_WIND_TEMP_MAX, Unit=°C, Disabled=FALSE)  // Motor: Limit temperature
          1210 = 2 (Name=MOTOR_TEMPMODEL_REFSENS, Disabled=FALSE)  // Motor: Temperature model: Reference sensor: Parameter-ID
          1211 = 0.2775 (Name=MOTOR_TEMPMODEL_RES1, Unit=K/W, Disabled=FALSE)  // Motor: Temperature model: Thermal resistance 1
          1212 = 17.226 (Name=MOTOR_TEMPMODEL_CAP1, Unit=Ws/K, Disabled=FALSE)  // Motor: Temperature model: Thermal capacity 1
          1213 = 0.4163 (Name=MOTOR_TEMPMODEL_RES2, Unit=K/W, Disabled=FALSE)  // Motor: Temperature model: Thermal resistance 2
          1214 = 0.348 (Name=MOTOR_TEMPMODEL_CAP2, Unit=Ws/K, Disabled=FALSE)  // Motor: Temperature model: Thermal capacity 2
          373 = 4 (Name=TEMP_MOTOR_MODEL_MODE, Disabled=FALSE)  // Motor: Temperature model: Mode
        Brake (Disabled=FALSE)
          42 = 0 (Name=MOTOR_BRAKE_CURR_RATED, Unit=A, Disabled=FALSE)  // Motor holding brake: Rated current
          43 = 0 (Name=MOTOR_BRAKE_TORQ_RATED, Unit=Nm, Disabled=FALSE)  // Motor holding brake: Rated torque
          44 = 0 (Name=MOTOR_BRAKE_ON_TIME, Unit=s, Disabled=FALSE)  // Motor holding brake: Engaging delay
          45 = 0 (Name=MOTOR_BRAKE_OFF_TIME, Unit=s, Disabled=FALSE)  // Motor holding brake: Release delay
        Temperature sensor (Disabled=FALSE)
          64 = 0 (Name=MOTOR_TEMPSENS_PAR1, Disabled=FALSE)  // Temperature sensor: Parameter 1
          65 = 0 (Name=MOTOR_TEMPSENS_PAR2, Disabled=FALSE)  // Temperature sensor: Parameter 2
          66 = 0 (Name=MOTOR_TEMPSENS_PAR3, Disabled=FALSE)  // Temperature sensor: Parameter 3
          67 = 0 (Name=MOTOR_TEMPSENS_PAR4, Disabled=FALSE)  // Temperature sensor: Parameter 4
          68 = 0 (Name=MOTOR_TEMPSENS_PAR5, Disabled=FALSE)  // Temperature sensor: Parameter 5
          69 = 0 (Name=MOTOR_TEMPSENS_PAR6, Disabled=FALSE)  // Temperature sensor: Parameter 6
          70 = 0 (Name=MOTOR_TEMPSENS_PAR7, Disabled=FALSE)  // Temperature sensor: Parameter 7
          71 = 0 (Name=MOTOR_TEMPSENS_PAR8, Disabled=FALSE)  // Temperature sensor: Parameter 8
          72 = 0 (Name=MOTOR_TEMPSENS_PAR9, Disabled=FALSE)  // Temperature sensor: Parameter 9
          73 = 0 (Name=MOTOR_TEMPSENS_PAR10, Disabled=FALSE)  // Temperature sensor: Parameter 10
        Encoder:
          652 = 0 (Name=MOTOR_ENCOD_ATTR, Disabled=FALSE)  // Motor: Encoder: Attribute
          1209 = 110 (Name=MOTOR_ENCOD_TEMP_LIM, Unit=°C, Disabled=FALSE)  // Motor: Encoder: Limit Temperature
          97 = ncLINMOT (Name=ENCOD_TYPE)  // Encoder1: Type
          109 = 16384 (Name=SCALE_ENCOD_INCR)  // Encoder1: Encoder scaling: increments per SCALE_ENCOD_MOTOR_REV motor revolutions
```

### Data object Logical/Real_Game/Motion/linearFWobj/linearFWi (Ax)

#### linearFWi.ax
```
InitParameter (Version=3.16.2)
  ACP10AXIS_typ:
    dig_in:
      level:
        reference = ncACTIV_HI
        pos_hw_end = ncACTIV_HI
        neg_hw_end = ncACTIV_HI
        trigger1 = ncACTIV_HI
        trigger2 = ncACTIV_HI
    encoder_if:
      parameter:
        count_dir = ncSTANDARD
        scaling:
          load:
            units = 200
            rev_motor = 1
    limit:
      parameter:
        v_pos = 30000.0
        v_neg = 30000.0
        a1_pos = 490000.0
        a2_pos = 490000.0
        a1_neg = 490000.0
        a2_neg = 490000.0
        t_jolt = 0.13
        t_in_pos = 0.0
        pos_sw_end = 881
        neg_sw_end = -821
        ds_warning = 200.0
        ds_stop = 200.0
        a_stop = 1.0E+30
        dv_stop = 0.0
        dv_stop_mode = ncOFF
    controller:
      mode = ncPOSITION + ncFF
      position:
        kv = 180.0
        tn = 0.0
        t_predict = 0.0004
        t_total = 0.0004
        p_max = 1.0E+30
        i_max = 0.0
      speed:
        kv = 0.2
        tn = 0.0
        t_filter = 0.0008
        isq_filter1:
          type = ncNOTCH
          a0 = 2328.77
          a1 = 2328.77
          b0 = 0.0
          b1 = 0.0
          b2 = 0.0
          c0_par_id = 0
          c1_par_id = 0
        isq_filter2:
          type = ncOFF
          a0 = 0.0
          a1 = 0.0
          b0 = 0.0
          b1 = 0.0
          b2 = 0.0
          c0_par_id = 0
          c1_par_id = 0
        isq_filter3:
          type = ncOFF
          a0 = 0.0
          a1 = 0.0
          b0 = 0.0
          b1 = 0.0
          b2 = 0.0
          c0_par_id = 0
          c1_par_id = 0
      uf:
        type = ncLINEAR
        auto_config = ncMOTOR_PAR
        u0 = 0.0
        un = 0.0
        fn = 50.0
        k_f_slip = 0.0
      ff:
        torque_load = 0.0
        torque_pos = 0.00691027
        torque_neg = 0.00674195
        kv_torque = 0.000864945
        inertia = 1.13117E-05
        t_filter_a = 0.0
    move:
      stop:
        parameter[0]:
          decel_ramp = ncA_LIMIT
          controller = ncON
        parameter[1]:
          decel_ramp = ncA_LIMIT
          controller = ncON
        parameter[2]:
          decel_ramp = ncA_LIMIT
          controller = ncON
        parameter[3]:
          decel_ramp = ncA_LIMIT
          controller = ncON
        quickstop:
          decel_ramp = ncA_LIMIT
        drive_error:
          decel_ramp = ncA_LIMIT
      homing:
        parameter:
          s = 880
          v_switch = 5000.0
          v_trigger = 5000.0
          a = 200000.0
          mode = ncBLOCK_TORQUE
          edge_sw = ncPOSITIVE
          start_dir = ncPOSITIVE
          trigg_dir = ncNEGATIVE
          ref_pulse = ncOFF
          fix_dir = ncOFF
          tr_s_block = 0.0
          torque_lim = 0.02
          ds_block = 0.0
          ds_stop = 1000.0
      basis:
        parameter:
          v_pos = 20000.0
          v_neg = 20000.0
          a1_pos = 400000.0
          a2_pos = 400000.0
          a1_neg = 400000.0
          a2_neg = 400000.0
    message:
      text:
        parameter:
          format = ncBREAK + ncZERO
          columns = 80
          data_modul = acp10etxen
```

### Package Logical/Real_Game/Motion/linearMDobj - linearMDobj

- Data object Logical/Real_Game/Motion/linearMDobj/linearMDa (Apt) (no source held here)

### Data object Logical/Real_Game/Motion/linearMDobj/linearMDi (Ax)

#### linearMDi.ax
```
InitParameter (Version=3.16.2)
  ACP10AXIS_typ:
    dig_in:
      level:
        reference = ncACTIV_HI
        pos_hw_end = ncACTIV_HI
        neg_hw_end = ncACTIV_HI
        trigger1 = ncACTIV_HI
        trigger2 = ncACTIV_HI
    encoder_if:
      parameter:
        count_dir = ncSTANDARD
        scaling:
          load:
            units = 200
            rev_motor = 1
    limit:
      parameter:
        v_pos = 30000.0
        v_neg = 30000.0
        a1_pos = 490000.0
        a2_pos = 490000.0
        a1_neg = 490000.0
        a2_neg = 490000.0
        t_jolt = 0.13
        t_in_pos = 0.0
        pos_sw_end = 571
        neg_sw_end = -551
        ds_warning = 200.0
        ds_stop = 200.0
        a_stop = 1.0E+30
        dv_stop = 0.0
        dv_stop_mode = ncOFF
    controller:
      mode = ncPOSITION + ncFF
      position:
        kv = 180.0
        tn = 0.0
        t_predict = 0.0004
        t_total = 0.0004
        p_max = 1.0E+30
        i_max = 0.0
      speed:
        kv = 0.2
        tn = 0.0
        t_filter = 0.0008
        isq_filter1:
          type = ncNOTCH
          a0 = 2328.77
          a1 = 2328.77
          b0 = 0.0
          b1 = 0.0
          b2 = 0.0
          c0_par_id = 0
          c1_par_id = 0
        isq_filter2:
          type = ncOFF
          a0 = 0.0
          a1 = 0.0
          b0 = 0.0
          b1 = 0.0
          b2 = 0.0
          c0_par_id = 0
          c1_par_id = 0
        isq_filter3:
          type = ncOFF
          a0 = 0.0
          a1 = 0.0
          b0 = 0.0
          b1 = 0.0
          b2 = 0.0
          c0_par_id = 0
          c1_par_id = 0
      uf:
        type = ncLINEAR
        auto_config = ncMOTOR_PAR
        u0 = 0.0
        un = 0.0
        fn = 50.0
        k_f_slip = 0.0
      ff:
        torque_load = 0.0
        torque_pos = 0.00691027
        torque_neg = 0.00674195
        kv_torque = 0.000864945
        inertia = 1.13117E-05
        t_filter_a = 0.0
    move:
      stop:
        parameter[0]:
          decel_ramp = ncA_LIMIT
          controller = ncON
        parameter[1]:
          decel_ramp = ncA_LIMIT
          controller = ncON
        parameter[2]:
          decel_ramp = ncA_LIMIT
          controller = ncON
        parameter[3]:
          decel_ramp = ncA_LIMIT
          controller = ncON
        quickstop:
          decel_ramp = ncA_LIMIT
        drive_error:
          decel_ramp = ncA_LIMIT
      homing:
        parameter:
          s = 570
          v_switch = 5000.0
          v_trigger = 5000.0
          a = 200000.0
          mode = ncBLOCK_TORQUE
          edge_sw = ncPOSITIVE
          start_dir = ncPOSITIVE
          trigg_dir = ncNEGATIVE
          ref_pulse = ncOFF
          fix_dir = ncOFF
          tr_s_block = 0.0
          torque_lim = 0.02
          ds_block = 0.0
          ds_stop = 1000.0
      basis:
        parameter:
          v_pos = 20000.0
          v_neg = 20000.0
          a1_pos = 400000.0
          a2_pos = 400000.0
          a1_neg = 400000.0
          a2_neg = 400000.0
    message:
      text:
        parameter:
          format = ncBREAK + ncZERO
          columns = 80
          data_modul = acp10etxen
```


- Data object Logical/Real_Game/Motion/rotDFobj/rotDFa (Apt) (no source held here)

- Data object Logical/Real_Game/Motion/rotDFobj/rotDFi (Ax) (no source held here)

- Data object Logical/Real_Game/Motion/rotDFVobj/rotDFVa (Apt) (no source held here)

- Data object Logical/Real_Game/Motion/rotDFVobj/rotDFVi (Vax) (no source held here)

- Data object Logical/Real_Game/Motion/rotGKobj/rotGKa (Apt) (no source held here)

- Data object Logical/Real_Game/Motion/rotGKobj/rotGKi (Ax) (no source held here)

### Package Logical/Real_Game/Motion/linDFobj - linDFobj

### Data object Logical/Real_Game/Motion/linDFobj/linDFa (Apt)

#### linDFa.apt
```
AcoposParameterTable:
  Root Parameters:
    linMot_PS01_23x80.xml:
      linMot__PS01_23x80.xml:
        LinMot: PS01-23x80/150x210  // Version: 1.1
          Motor (Disabled=FALSE)
            30 = 0x0002 (Name=MOTOR_TYPE, Disabled=FALSE)  // Motor: Type
            31 = 0x0203 (Name=MOTOR_COMPATIBILITY, Disabled=FALSE)  // Motor: Software compatibility
            46 = 1 (Name=MOTOR_WIND_CONNECT, Disabled=FALSE)  // Motor: Winding connection
            47 = 1 (Name=MOTOR_POLEPAIRS, Disabled=FALSE)  // Motor: Number of pole-pairs
            1208 = 2 (Name=MOTOR_NUM_PHASES)  // Motor: Number of motor phases
            48 = 72 (Name=MOTOR_VOLTAGE_RATED, Unit=V, Disabled=FALSE)  // Motor: Rated voltage
            49 = 5.209 (Name=MOTOR_VOLTAGE_CONST, Unit=mV*min, Disabled=FALSE)  // Motor: Voltage constant
            51 = 18000 (Name=MOTOR_SPEED_MAX, Unit=1/min, Disabled=FALSE)  // Motor: Maximum speed
            54 = 0.14 (Name=MOTOR_TORQ_MAX, Unit=Nm, Disabled=FALSE)  // Motor: Peak torque
            55 = 0.035 (Name=MOTOR_TORQ_CONST, Unit=Nm/A, Disabled=FALSE)  // Motor: Torque constant
            58 = 4 (Name=MOTOR_CURR_MAX, Unit=A, Disabled=FALSE)  // Motor: Peak current
            60 = 12.5 (Name=MOTOR_STATOR_RESISTANCE, Unit=Ohm, Disabled=FALSE)  // Motor: Stator resistance
            61 = 0.0014 (Name=MOTOR_STATOR_INDUCTANCE, Unit=Henry, Disabled=FALSE)  // Motor: Stator inductance
            62 = 0.0000027 (Name=MOTOR_INERTIA, Unit=kgmp, Disabled=FALSE)  // Motor: Moment of inertia
            63 = 1.5707963 (Name=MOTOR_COMMUT_OFFSET, Unit=rad, Disabled=FALSE)  // Motor: Commutation offset
            276 = 4 (Name=PHASING_MODE, Disabled=FALSE)  // Motor: Phasing: Mode
          50 = 18000 (Name=MOTOR_SPEED_RATED, Unit=1/min, Disabled=FALSE)  // Motor: Rated speed
          Temperature model (Disabled=FALSE)
            56 = 0.82 (Name=MOTOR_CURR_STALL, Unit=A, Disabled=FALSE)  // Motor: Stall current
            57 = 0.82 (Name=MOTOR_CURR_RATED, Unit=A, Disabled=FALSE)  // Motor: Rated current
            52 = 0.03 (Name=MOTOR_TORQ_STALL, Unit=Nm, Disabled=FALSE)  // Motor: Stall torque
            53 = 0.03 (Name=MOTOR_TORQ_RATED, Unit=Nm, Disabled=FALSE)  // Motor: Rated torque
            59 = 0.11 (Name=MOTOR_WIND_CROSS_SECT, Unit=mmp, Disabled=FALSE)  // Motor: Line cross section
            849 = 135.72 (Name=MOTOR_TAU_THERM, Unit=s, Disabled=FALSE)  // Motor: Thermal time constant
            74 = 110 (Name=MOTOR_WIND_TEMP_MAX, Unit=°C, Disabled=FALSE)  // Motor: Limit temperature
            1210 = 2 (Name=MOTOR_TEMPMODEL_REFSENS, Disabled=FALSE)  // Motor: Temperature model: Reference sensor: Parameter-ID
            1211 = 0.2775 (Name=MOTOR_TEMPMODEL_RES1, Unit=K/W, Disabled=FALSE)  // Motor: Temperature model: Thermal resistance 1
            1212 = 17.226 (Name=MOTOR_TEMPMODEL_CAP1, Unit=Ws/K, Disabled=FALSE)  // Motor: Temperature model: Thermal capacity 1
            1213 = 0.4163 (Name=MOTOR_TEMPMODEL_RES2, Unit=K/W, Disabled=FALSE)  // Motor: Temperature model: Thermal resistance 2
            1214 = 0.348 (Name=MOTOR_TEMPMODEL_CAP2, Unit=Ws/K, Disabled=FALSE)  // Motor: Temperature model: Thermal capacity 2
            373 = 4 (Name=TEMP_MOTOR_MODEL_MODE, Disabled=FALSE)  // Motor: Temperature model: Mode
          Brake (Disabled=FALSE)
            42 = 0 (Name=MOTOR_BRAKE_CURR_RATED, Unit=A, Disabled=FALSE)  // Motor holding brake: Rated current
            43 = 0 (Name=MOTOR_BRAKE_TORQ_RATED, Unit=Nm, Disabled=FALSE)  // Motor holding brake: Rated torque
            44 = 0 (Name=MOTOR_BRAKE_ON_TIME, Unit=s, Disabled=FALSE)  // Motor holding brake: Engaging delay
            45 = 0 (Name=MOTOR_BRAKE_OFF_TIME, Unit=s, Disabled=FALSE)  // Motor holding brake: Release delay
          Temperature sensor (Disabled=FALSE)
            64 = 0 (Name=MOTOR_TEMPSENS_PAR1, Disabled=FALSE)  // Temperature sensor: Parameter 1
            65 = 0 (Name=MOTOR_TEMPSENS_PAR2, Disabled=FALSE)  // Temperature sensor: Parameter 2
            66 = 0 (Name=MOTOR_TEMPSENS_PAR3, Disabled=FALSE)  // Temperature sensor: Parameter 3
            67 = 0 (Name=MOTOR_TEMPSENS_PAR4, Disabled=FALSE)  // Temperature sensor: Parameter 4
            68 = 0 (Name=MOTOR_TEMPSENS_PAR5, Disabled=FALSE)  // Temperature sensor: Parameter 5
            69 = 0 (Name=MOTOR_TEMPSENS_PAR6, Disabled=FALSE)  // Temperature sensor: Parameter 6
            70 = 0 (Name=MOTOR_TEMPSENS_PAR7, Disabled=FALSE)  // Temperature sensor: Parameter 7
            71 = 0 (Name=MOTOR_TEMPSENS_PAR8, Disabled=FALSE)  // Temperature sensor: Parameter 8
            72 = 0 (Name=MOTOR_TEMPSENS_PAR9, Disabled=FALSE)  // Temperature sensor: Parameter 9
            73 = 0 (Name=MOTOR_TEMPSENS_PAR10, Disabled=FALSE)  // Temperature sensor: Parameter 10
          Encoder:
            652 = 0 (Name=MOTOR_ENCOD_ATTR, Disabled=FALSE)  // Motor: Encoder: Attribute
            1209 = 110 (Name=MOTOR_ENCOD_TEMP_LIM, Unit=°C, Disabled=FALSE)  // Motor: Encoder: Limit Temperature
            97 = ncLINMOT (Name=ENCOD_TYPE)  // Encoder1: Type
            109 = 16384 (Name=SCALE_ENCOD_INCR)  // Encoder1: Encoder scaling: increments per SCALE_ENCOD_MOTOR_REV motor revolutions
```

### Data object Logical/Real_Game/Motion/linDFobj/linDFi (Ax)

#### linDFi.ax
```
InitParameter (Version=3.16.2)
  ACP10AXIS_typ:
    dig_in:
      level:
        reference = ncACTIV_HI
        pos_hw_end = ncACTIV_HI
        neg_hw_end = ncACTIV_HI
        trigger1 = ncACTIV_HI
        trigger2 = ncACTIV_HI
    encoder_if:
      parameter:
        count_dir = ncSTANDARD
        scaling:
          load:
            units = 200
            rev_motor = 1
    limit:
      parameter:
        v_pos = 30000.0
        v_neg = 30000.0
        a1_pos = 490000.0
        a2_pos = 490000.0
        a1_neg = 490000.0
        a2_neg = 490000.0
        t_jolt = 0.13
        t_in_pos = 0.0
        pos_sw_end = 1081
        neg_sw_end = -981
        ds_warning = 200.0
        ds_stop = 200.0
        a_stop = 1.0E+30
        dv_stop = 0.0
        dv_stop_mode = ncOFF
    controller:
      mode = ncPOSITION + ncFF
      position:
        kv = 180.0
        tn = 0.0
        t_predict = 0.0004
        t_total = 0.0004
        p_max = 1.0E+30
        i_max = 0.0
      speed:
        kv = 0.2
        tn = 0.0
        t_filter = 0.0008
        isq_filter1:
          type = ncNOTCH
          a0 = 2328.77
          a1 = 2328.77
          b0 = 0.0
          b1 = 0.0
          b2 = 0.0
          c0_par_id = 0
          c1_par_id = 0
        isq_filter2:
          type = ncOFF
          a0 = 0.0
          a1 = 0.0
          b0 = 0.0
          b1 = 0.0
          b2 = 0.0
          c0_par_id = 0
          c1_par_id = 0
        isq_filter3:
          type = ncOFF
          a0 = 0.0
          a1 = 0.0
          b0 = 0.0
          b1 = 0.0
          b2 = 0.0
          c0_par_id = 0
          c1_par_id = 0
      uf:
        type = ncLINEAR
        auto_config = ncMOTOR_PAR
        u0 = 0.0
        un = 0.0
        fn = 50.0
        k_f_slip = 0.0
      ff:
        torque_load = 0.0
        torque_pos = 0.00691027
        torque_neg = 0.00674195
        kv_torque = 0.000864945
        inertia = 1.13117E-05
        t_filter_a = 0.0
    move:
      stop:
        parameter[0]:
          decel_ramp = ncA_LIMIT
          controller = ncON
        parameter[1]:
          decel_ramp = ncA_LIMIT
          controller = ncON
        parameter[2]:
          decel_ramp = ncA_LIMIT
          controller = ncON
        parameter[3]:
          decel_ramp = ncA_LIMIT
          controller = ncON
        quickstop:
          decel_ramp = ncA_LIMIT
        drive_error:
          decel_ramp = ncA_LIMIT
      homing:
        parameter:
          s = 1080
          v_switch = 5000.0
          v_trigger = 5000.0
          a = 200000.0
          mode = ncBLOCK_TORQUE
          edge_sw = ncPOSITIVE
          start_dir = ncPOSITIVE
          trigg_dir = ncNEGATIVE
          ref_pulse = ncOFF
          fix_dir = ncOFF
          tr_s_block = 0.0
          torque_lim = 0.02
          ds_block = 0.0
          ds_stop = 1200.0
      basis:
        parameter:
          v_pos = 20000.0
          v_neg = 20000.0
          a1_pos = 400000.0
          a2_pos = 400000.0
          a1_neg = 400000.0
          a2_neg = 400000.0
    message:
      text:
        parameter:
          format = ncBREAK + ncZERO
          columns = 80
          data_modul = acp10etxen
```

### Package Logical/Real_Game/Motion/linDFVobj - linDFVobj

- Data object Logical/Real_Game/Motion/linDFVobj/linDFVa (Apt) (no source held here)

### Data object Logical/Real_Game/Motion/linDFVobj/linDFVi (Vax)

- linDFVi.vax (not shown)

### Package Logical/Real_Game/Motion/linGKobj - linGKobj

- Data object Logical/Real_Game/Motion/linGKobj/linGKa (Apt) (no source held here)

### Data object Logical/Real_Game/Motion/linGKobj/linGKi (Ax)

#### linGKi.ax
```
InitParameter (Version=3.16.2)
  ACP10AXIS_typ:
    dig_in:
      level:
        reference = ncACTIV_HI
        pos_hw_end = ncACTIV_HI
        neg_hw_end = ncACTIV_HI
        trigger1 = ncACTIV_HI
        trigger2 = ncACTIV_HI
    encoder_if:
      parameter:
        count_dir = ncSTANDARD
        scaling:
          load:
            units = 200
            rev_motor = 1
    limit:
      parameter:
        v_pos = 30000.0
        v_neg = 30000.0
        a1_pos = 490000.0
        a2_pos = 490000.0
        a1_neg = 490000.0
        a2_neg = 490000.0
        t_jolt = 0.13
        t_in_pos = 0.0
        pos_sw_end = 821
        neg_sw_end = -931
        ds_warning = 200.0
        ds_stop = 200.0
        a_stop = 1.0E+30
        dv_stop = 0.0
        dv_stop_mode = ncOFF
    controller:
      mode = ncPOSITION + ncFF
      position:
        kv = 180.0
        tn = 0.0
        t_predict = 0.0004
        t_total = 0.0004
        p_max = 1.0E+30
        i_max = 0.0
      speed:
        kv = 0.2
        tn = 0.0
        t_filter = 0.0008
        isq_filter1:
          type = ncNOTCH
          a0 = 2328.77
          a1 = 2328.77
          b0 = 0.0
          b1 = 0.0
          b2 = 0.0
          c0_par_id = 0
          c1_par_id = 0
        isq_filter2:
          type = ncOFF
          a0 = 0.0
          a1 = 0.0
          b0 = 0.0
          b1 = 0.0
          b2 = 0.0
          c0_par_id = 0
          c1_par_id = 0
        isq_filter3:
          type = ncOFF
          a0 = 0.0
          a1 = 0.0
          b0 = 0.0
          b1 = 0.0
          b2 = 0.0
          c0_par_id = 0
          c1_par_id = 0
      uf:
        type = ncLINEAR
        auto_config = ncMOTOR_PAR
        u0 = 0.0
        un = 0.0
        fn = 50.0
        k_f_slip = 0.0
      ff:
        torque_load = 0.0
        torque_pos = 0.00691027
        torque_neg = 0.00674195
        kv_torque = 0.000864945
        inertia = 1.13117E-05
        t_filter_a = 0.0
    move:
      stop:
        parameter[0]:
          decel_ramp = ncA_LIMIT
          controller = ncON
        parameter[1]:
          decel_ramp = ncA_LIMIT
          controller = ncON
        parameter[2]:
          decel_ramp = ncA_LIMIT
          controller = ncON
        parameter[3]:
          decel_ramp = ncA_LIMIT
          controller = ncON
        quickstop:
          decel_ramp = ncA_LIMIT
        drive_error:
          decel_ramp = ncA_LIMIT
      homing:
        parameter:
          s = 820
          v_switch = 5000.0
          v_trigger = 5000.0
          a = 200000.0
          mode = ncBLOCK_TORQUE
          edge_sw = ncPOSITIVE
          start_dir = ncPOSITIVE
          trigg_dir = ncNEGATIVE
          ref_pulse = ncOFF
          fix_dir = ncOFF
          tr_s_block = 0.0
          torque_lim = 0.02
          ds_block = 0.0
          ds_stop = 1000.0
      basis:
        parameter:
          v_pos = 20000.0
          v_neg = 20000.0
          a1_pos = 400000.0
          a2_pos = 400000.0
          a1_neg = 400000.0
          a2_neg = 400000.0
    message:
      text:
        parameter:
          format = ncBREAK + ncZERO
          columns = 80
          data_modul = acp10etxen
```

### Program Logical/Real_Game/Technology/table_football (ANSIC) - Roman Parák program for real game.

#### mapp.h
```c
/*********************************************************************************************
* B&R Automation - Perfection in Automation (https://www.br-automation.com)
    ******************************************************************************************
    * Program 	    : Master's Thesis - Soccer Table (Table Football - real game)
    * Author  	    : Roman Parak
    * Created 	    : date ...
	* University    : Brno University of Technology(BUT)
	* Faculty       : Faculty of Mechanical Engineering(FME)
	* Study Program : Applied Computer Science and Control
	* Institute     : Institute of Automation and Computer Science
**********************************************************************************************
* Implementation OF PROGRAM table_football(Real_Game/Technolog/table_football/Functions/mapp.h)
**********************************************************************************************/

/*************************** LIBRARIES *********************************/
#include <bur/plc.h>
#include <bur/plctypes.h>
#include <AsString.h>
#include <standard.h>
#include <AsWStr.h>
#include <stdio.h>
#include <math.h>

#ifdef _DEFAULT_INCLUDES
    #include <AsDefault.h>
#endif

/**********************************************************************************************************/
/************************************** FUNCTIONS & FUNCTIONS BLOCKS **************************************/
/**********************************************************************************************************/
void start_axesBasic(USINT num_ofAxes,struct MpAxisBasic* axis_linear,struct MpAxisBasic* axis_rotary){
    int i;
    // Axis Basic
    // function to start the individual axes
    // the cycle is carried out through number of axes
    for(i = 0; i <= num_ofAxes - 1; i++){
        // mapp axis basic
        MpAxisBasic(&axis_linear[i]);
        MpAxisBasic(&axis_rotary[i]);
    }
}

void start_axesCyclic(USINT num_ofAxes,struct MpAxisCyclicSet* cyclic_linear,struct MpAxisCyclicSet* cyclic_rotary){
    int i;
    // Axis Cyclic Set
    // function to start the individual axes
    // the cycle is carried out through number of axes
    for(i = 0; i <= num_ofAxes - 1; i++){
        // mapp axis cyclic set
        MpAxisCyclicSet(&cyclic_linear[i]);
        MpAxisCyclicSet(&cyclic_rotary[i]);
    }
}

struct axesAcopos get_axisParam(int idx_ofIteration){
    // input into the function is number of iteration(in the init part)
    // create auxiliary structures and enumeration type(for state machine)
    struct axesAcopos a;
    typedef enum {aNUM1 = 0, aNUM2, aNUM3, aNUM4}wState_ofAxes;
    wState_ofAxes new_idx; // initialize state machine
    new_idx = idx_ofIteration;
    // gradually into the state machine loading indexes from initialization part
    // and this run the function blocks
    // each state of machine has initialization both engines linear and rotary, on its own axis
    // output of this function is structure, that has two parameters(linear,rotary axis)
    switch(new_idx){
        case aNUM1:
            // goalkeeper
            a.linear = &linGK;
            a.rotary = &rotGK;
            return a;
            break;
        case aNUM2:
            // defender
            a.linear = &linDF;
            a.rotary = &rotDF;
            return a;
            break;
        case aNUM3:
            // midfielder
            a.linear = &linearMD;
            a.rotary = &rotaryMD;
            return a;
            break;
        case aNUM4:
            // forward
            a.linear = &linearFW;
            a.rotary = &rotaryFW;
			return a;
            break;
    }
}

void start_cs(USINT num_ofAxes,struct MpAxisCyclicSet* cyclic_linear,struct MpAxisCyclicSet* cyclic_rotary){

	switch(num_ofAxes){
		case 1:
			{
				cyclic_linear[0].CyclicPosition = 1;
				cyclic_rotary[0].CyclicPosition = 1;
			}
			break;
		case 2:
			{
				cyclic_linear[0].CyclicPosition = 1;
				cyclic_linear[1].CyclicPosition = 1;
				cyclic_rotary[0].CyclicPosition = 1;
				cyclic_rotary[1].CyclicPosition = 1;

			}
			break;
		case 3:
			{
				cyclic_linear[0].CyclicPosition = 1;
				cyclic_linear[1].CyclicPosition = 1;
				cyclic_linear[2].CyclicPosition = 1;
				cyclic_rotary[0].CyclicPosition = 1;
				cyclic_rotary[1].CyclicPosition = 1;
				cyclic_rotary[2].CyclicPosition = 1;
			}
			break;
		case 4:
			{
				cyclic_linear[0].CyclicPosition = 1;
				cyclic_linear[1].CyclicPosition = 1;
				cyclic_linear[2].CyclicPosition = 1;
				cyclic_linear[3].CyclicPosition = 1;
				cyclic_rotary[0].CyclicPosition = 1;
				cyclic_rotary[1].CyclicPosition = 1;
				cyclic_rotary[2].CyclicPosition = 1;
				cyclic_rotary[3].CyclicPosition = 1;
			}
			break;
	}// end switch

}
```
